FUNCTION_BLOCK FB_VariableMotor IMPLEMENTS I_Motor

VAR
	bRunning : BOOL;
END_VAR

{warning 'add method implementation '}
METHOD Start : BOOL
Start := bRunning := TRUE;
END_METHOD

{warning 'add method implementation '}
METHOD Stop : BOOL
bRunning := FALSE;
Stop := NOT bRunning;
END_METHOD

END_FUNCTION_BLOCK

(* stored: Version 1.1.0.1, ProductVersion 3.1.4024.16
   POU FB_VariableMotor: Id {ad2eb346-c54c-4c8d-96ba-c5d7217fbd90}, SpecialFunc None
   Method Start: Id {ebceca45-5ab8-42b2-be82-2d157e02b4d1}
   Method Stop: Id {2cecf2fe-7547-4c68-bee1-c640df9eb39d} *)
